FUNCTION_BLOCK FB_Blink
VAR_INPUT
	timeOn:TIME:=T#300MS;
	timeOff:TIME:=T#500MS;
END_VAR
VAR_OUTPUT
	bOutput: BOOL;
END_VAR
VAR
	timer:TON;
END_VAR

timer(IN:= NOT timer.Q);
IF timer.Q THEN
	IF bOutput THEN
		timer.PT:=timeOff;
	ELSE
		timer.PT:=timeOn;	
	END_IF
	bOutput:= NOT bOutput;
END_IF

END_FUNCTION_BLOCK

(* stored: Version 1.1.0.1, ProductVersion 3.1.4024.12
   POU FB_Blink: Id {7f6ddd49-071f-4e9a-b350-8602ca22eef3}, SpecialFunc None *)
